FUNCTION_BLOCK FB_HaltNC IMPLEMENTS I_Halt
VAR_INPUT
    {attribute 'no_copy'}
    AxisRef : REFERENCE TO AXIS_REF;
    fbMcHalt 		: MC_Halt;
    bExecute :BOOL;
    fDeceleration : LREAL;
    fJerk :LREAL;
    eBufferMode : MC_BufferMode := MC_BufferMode.MC_Aborting;
    bError : BOOL;
    bBusy : BOOL;
    bDone : BOOL;
    nErrorID : UDINT;
    sMessage : T_MAXSTRING;
    rtDone : R_TRIG;
END_VAR
VAR_OUTPUT
END_VAR
VAR
END_VAR

THIS^.fbMcHalt(
    Axis := THIS^.AxisRef,
    Execute := THIS^.bExecute,
    Deceleration := THIS^.fDeceleration,
    Jerk := THIS^.fJerk,
    BufferMode := THIS^.eBufferMode,
    Done =>THIS^.bDone,
    Busy => THIS^.bBusy,
    CommandAborted => ,
    Error => THIS^.bError,
    ErrorID => THIS^.nErrorID
);

rtDone(CLK:=bDone);
IF  rtDone.Q THEN
    THIS^.bExecute := FALSE;
END_IF

{warning 'add property implementation'}
PROPERTY ExecHalt : BOOL
SET
THIS^.bExecute :=  ExecHalt;
END_SET
END_PROPERTY

//FB_Init is always available implicitly and it is used primarily for initialization.
//The return value is not evaluated. For a specific influence, you can also declare the
//methods explicitly and provide additional code there with the standard initialization
//code. You can evaluate the return value.
METHOD FB_Init: BOOL
VAR_INPUT
    bInitRetains: BOOL; // TRUE: the retain variables are initialized (reset warm / reset cold)
    bInCopyCode: BOOL;  // TRUE: the instance will be copied to the copy code afterward (online change)
    AxisRef : REFERENCE TO AXIS_REF;
END_VAR
THIS^.AxisRef REF= AxisRef;
END_METHOD

METHOD Halt
VAR_INPUT
    Execute	: BOOL;
    Deceleration	: LREAL := 0;
    Jerk	: LREAL := 0;
    BufferMode	: MC_BufferMode := .MC_BufferMode.MC_Aborting;
END_VAR
THIS^.bExecute :=  Execute;
THIS^.fDeceleration := Deceleration;
THIS^.fJerk := Jerk;
THIS^.eBufferMode := BufferMode;
END_METHOD

PROPERTY HaltBufferMode : Tc2_MC2.MC_BufferMode
SET
eBufferMode := HaltBufferMode;
END_SET
END_PROPERTY

{warning 'add property implementation'}
PROPERTY HaltBusy : BOOL
GET
HaltBusy := bBusy;
END_GET
END_PROPERTY

{warning 'add property implementation'}
PROPERTY HaltDeceleration : LREAL
SET
THIS^.fDeceleration := HaltDeceleration;
END_SET
END_PROPERTY

PROPERTY HaltDone : BOOL
GET
HaltDone := bDone;
END_GET
END_PROPERTY

{warning 'add property implementation'}
PROPERTY HaltError : BOOL
GET
HaltError := bError;
END_GET
END_PROPERTY

{warning 'add property implementation'}
PROPERTY HaltErrorID : UDINT
GET
HaltErrorID := nErrorID;
END_GET
END_PROPERTY

PROPERTY HaltJerk : LREAL
SET
fJerk := HaltJerk;
END_SET
END_PROPERTY

END_FUNCTION_BLOCK

(* stored: Version 1.1.0.1
   POU FB_HaltNC: Id {c033f4f8-0634-4c06-a30f-6a4c2be036bc}, SpecialFunc None
   Property ExecHalt: Id {b029dd2e-4ddf-4863-82b3-8648d81b0ad5}
   Set Set: Id {e67d86a9-bf4d-478f-a33b-2d93cc2ff9cf}
   Method FB_Init: Id {18cebc01-b938-405d-8b68-4f57807b525a}
   Method Halt: Id {7d31f5d0-f1cb-401e-ae13-f0dc85da0693}
   Property HaltBufferMode: Id {7337b28e-2d64-4cf3-a38d-55c6ef1e0217}
   Set Set: Id {4fa05682-b652-4121-b44d-4a8b2a3bc935}
   Property HaltBusy: Id {2883f0f4-4b95-4139-8a36-d2b2f3dcc31b}
   Get Get: Id {5b77bc7a-e864-4e13-ae17-e0016b7d86c8}
   Property HaltDeceleration: Id {53e71343-314a-4971-812b-de31ec077725}
   Set Set: Id {8aa39272-ea7c-4c8a-88cc-b19176760b77}
   Property HaltDone: Id {be7dfb74-7669-4f3f-93f0-cda14723d1f0}
   Get Get: Id {0f32e8ae-880b-42bd-b635-3e016d1c20ba}
   Property HaltError: Id {45d4ccdb-82f3-4b2c-ae9a-f7a118e27ac3}
   Get Get: Id {bbf7cb10-277f-4907-9b37-03e01cec3c96}
   Property HaltErrorID: Id {336845aa-0c0a-4c8a-b21e-bc9fafd47d20}
   Get Get: Id {d0994f69-d16e-4cfd-8b2d-204ea0c00d54}
   Property HaltJerk: Id {ccf57f45-64a9-413b-b5e8-74695a1b4351}
   Set Set: Id {5532a8e1-15d6-4ddf-bcad-8d399efcf14b} *)
